PROGRAM MAIN
VAR
	
    {attribute 'pytmc' := '
      pv: VCN:TEST:01
    '}
	fbVCN590 : FB_VCN_VAT590; // Variable leak valve VAT590 function block
	
	stVG : ST_VG;
    {attribute 'pytmc' := '
      pv: GHC:TEST
    '}
	fbIE514 : FB_IE514;
	
    {attribute 'pytmc' := '
      pv: GCC:TEST:02
    '}
	fbMX7M : FB_MX7M;
	
    {attribute 'pytmc' := '
      pv: GHC:TEST:03
    '}
	fbIMG401 : FB_IMG401;
	
	rPiraniPressure : REAL := 1E-4;
	bPressOK : BOOL := TRUE;
END_VAR

stVG.xPRESS_OK := bPressOK;
stVG.rPress := rPiraniPressure;
stVG.eState := ValidLo;
stVG.xAT_VAC := TRUE;

fbIMG401.M_SetBits(30518);
fbIMG401(PG := stVG);

fbVCN590(bExtIlkOK := TRUE, IG := fbIMG401.IG);

//fbIE514(PG := stVG);

//fbMX7M(PG := stVG);

END_PROGRAM

(* stored: Version 1.1.0.1, ProductVersion 3.1.4022.18
   POU MAIN: Id {e705ade6-0f0a-4b24-98f0-3b81c602a7eb}, SpecialFunc None *)
